// TIA Portal V17 export
// export: Created 2024-09-03T21:55:05.0012998Z, ExportSetting WithDefaults, DisplayName Totally Integrated Automation Portal, DisplayVersion V17 Update 7, DisplayName TIA Portal Openness, DisplayVersion V17 Update 7, DisplayName TIA Portal Version Control Interface, DisplayVersion V17, DisplayName SINAMICS Startdrive Advanced, DisplayVersion V17 SP2, DisplayName SINAMICS Startdrive G110M, G120, G120C, G120D, G120P, G115D, DisplayVersion V17 SP2, DisplayName SINAMICS Startdrive G130, G150, S120, S150, SINAMICS MV, S210, DisplayVersion V17 SP2, DisplayName STEP 7 Professional, DisplayVersion V17 Update 7, DisplayName STEP 7 Safety, DisplayVersion V17 Update 6, DisplayName WinCC Advanced / Unified PC, DisplayVersion V17 Update 7
TYPE "UDT_Servo"
// stored: IsFailsafeCompliant false
   STRUCT
      ModePos : Int;
      EnableAxis : Bool;
      CancelTraversing : Bool;
      IntermediateStop : Bool;
      Positive : Bool;
      Negative : Bool;
      Jog1 : Bool;
      Jog2 : Bool;
      FlyRef : Bool;
      AckError : Bool;
      ExecuteMode : Bool;
      Position : DInt;
      Velocity : DInt;
      OverV : Int;
      OverAcc : Int;
      OverDec : Int;
      AxisEnabled : Bool;
      AxisPosOk : Bool;
      AxisSpFixed : Bool;
      AxisRef : Bool;
      AxisWarn : Bool;
      AxisError : Bool;
      Lockout : Bool;
      ActVelocity : DInt;
      ActPosition : DInt;
      ActMode : Int;
      EPosZSW1 : Word;
      EPosZSW2 : Word;
      ActWarn : Word;
      ActFault : Word;
      Error : Bool;
      Status : Word;
      DiagID : Word;
      data : Struct
         zones : Struct
            inST3jig : Bool;
            inOKpos : Bool;
            inNOKpos : Bool;
            outOfST3zone : Bool;
            outOfOKposZone : Bool;
         END_STRUCT;
      END_STRUCT;
   END_STRUCT;
END_TYPE
